FUNCTION_BLOCK FB_CsvFileWriter IMPLEMENTS I_FileWriter

VAR
	sMessageString : STRING;
	eWriteState : (FILE_OPEN_TRIGGER, FILE_OPEN, WAIT_FOR_EVENT, WRITE_EVENT_TRIGGER, WRITE_EVENT,FILE_CLOSE_TRIGGER, FILE_CLOSE, ERROR );
	fbFileOpen : FB_FileOpen := (sPathName := 'C:\Users\kameshwaran.k\OneDrive - InTimeTec Visionsoft Pvt. Ltd.,\Documents/Event.txt', nMode := FOPEN_MODEAPPEND OR FOPEN_MODETEXT);
	fbFilePuts : FB_FilePuts;
	fbFileClose : FB_FileClose;
	sCsvString : T_MaxString ;
END_VAR

CASE eWriteState OF
	FILE_OPEN_TRIGGER:
	fbFileOpen(bExecute := TRUE);
	eWriteState := FILE_OPEN;
	
	FILE_OPEN:
	fbFileOpen(bExecute := FALSE);
	IF fbFileOpen.bError THEN
		eWriteState := ERROR;
		ELSIF NOT fbFileOpen.bBusy AND fbFileOpen.hFile <> 0 THEN
			eWriteState := WAIT_FOR_EVENT;
	END_IF
	WAIT_FOR_EVENT:	
	//No logic 
	
	WRITE_EVENT_TRIGGER:
	sCsvString := ConvertString(sString := sMessageString);
	fbFilePuts(bExecute := TRUE, sLine := sCsvString, hFile := fbFileOpen.hFile);
	eWriteState := WRITE_EVENT;
	
	WRITE_EVENT:
	fbFilePuts(bExecute := FALSE);
	IF fbFilePuts.bError THEN
		eWriteState := ERROR;
		ELSIF NOT fbFilePuts.bBusy THEN
			eWriteState := FILE_CLOSE_TRIGGER;
			
	END_IF
	
	FILE_CLOSE_TRIGGER:
	fbFileClose(bExecute := TRUE, hFile := fbFileOpen.hFile);
	eWriteState := FILE_CLOSE;
	
	FILE_CLOSE:
	fbFileClose(bExecute := FALSE);
	IF fbFileClose.bError THEN
		eWriteState := ERROR;
		ELSIF NOT fbFileClose.bBusy THEN
			eWriteState := FILE_OPEN_TRIGGER;
	END_IF
	ERROR:
END_CASE

METHOD PRIVATE ConvertString : T_MaxString
VAR_INPUT
	sString : STRING;
END_VAR
ConvertString := CONCAT(STR1 := sString , STR2 := '$n');
END_METHOD

{warning 'add method implementation '}
METHOD WriteEvent : BOOL
VAR_INPUT
	sMessage : STRING ;
END_VAR
IF eWriteState = WAIT_FOR_EVENT THEN
	eWriteState := WRITE_EVENT_TRIGGER;
	sMessageString := sMessage;
END_IF
END_METHOD

END_FUNCTION_BLOCK

(* stored: Version 1.1.0.1, ProductVersion 3.1.4024.16
   POU FB_CsvFileWriter: Id {985302f9-bc50-42eb-a1b8-48062d78235a}, SpecialFunc None
   Method ConvertString: Id {d26c4cce-9016-4b50-991e-96f9e3f59249}
   Method WriteEvent: Id {49f2f820-eea2-41fa-b661-c20737d4db05} *)
